// TIA Portal V17 export
// export: Created 2024-06-16T17:47:20.4638642Z, ExportSetting WithDefaults, DisplayName Totally Integrated Automation Portal, DisplayVersion V17, DisplayName TIA Portal Openness, DisplayVersion V17, DisplayName TIA Portal Version Control Interface, DisplayVersion V17, DisplayName STEP 7 Professional, DisplayVersion V17, DisplayName STEP 7 Safety, DisplayVersion V17, DisplayName WinCC Professional, DisplayVersion V17
FUNCTION "Manager" : Void   // FC1, LAD
{ S7_Optimized_Access := 'TRUE' }
VERSION : 0.1
// stored: AutoNumber false, IsIECCheckEnabled false, SetENOAutomatically false, UDAEnableTagReadback false
BEGIN

REGION Network 1
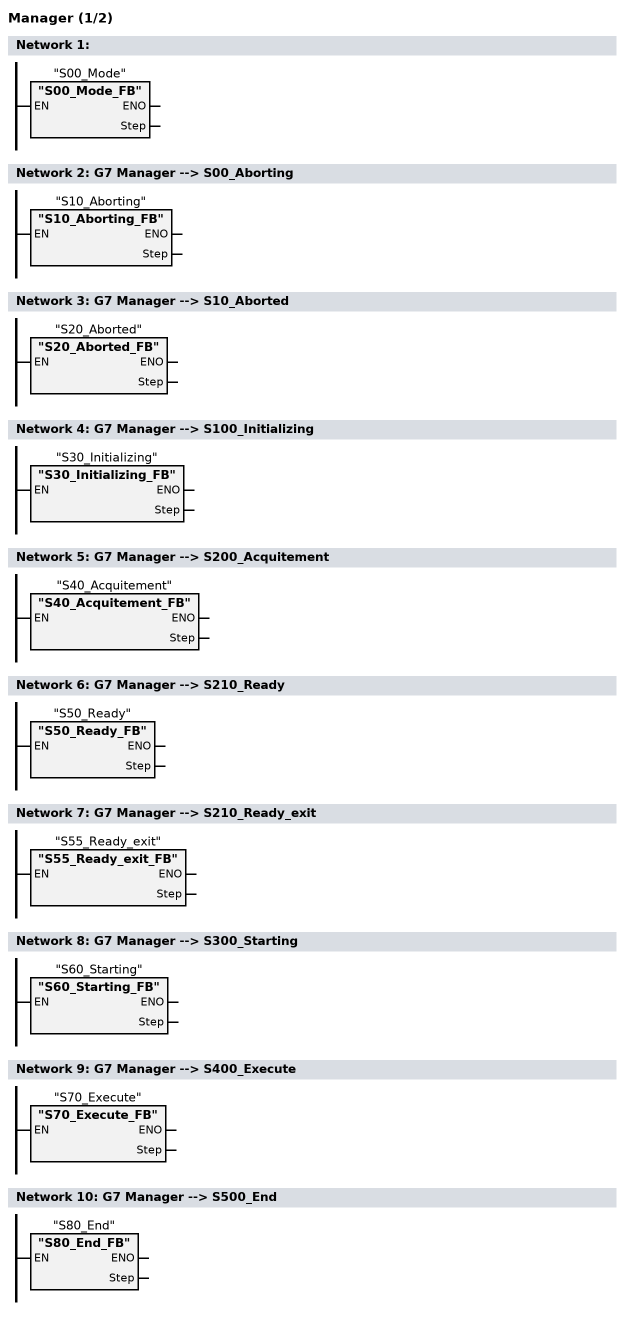
   RUNG wire#powerrail
      "S00_Mode"("Step" =>)
   END_RUNG
   // the same network as SCL:
   "S00_Mode"();   // "S00_Mode_FB"
END_REGION

REGION Network 2: G7 Manager --> S00_Aborting
   RUNG wire#powerrail
      "S10_Aborting"("Step" =>)
   END_RUNG
   // the same network as SCL:
   "S10_Aborting"();   // "S10_Aborting_FB"
END_REGION

REGION Network 3: G7 Manager --> S10_Aborted
   RUNG wire#powerrail
      "S20_Aborted"("Step" =>)
   END_RUNG
   // the same network as SCL:
   "S20_Aborted"();   // "S20_Aborted_FB"
END_REGION

REGION Network 4: G7 Manager --> S100_Initializing
   RUNG wire#powerrail
      "S30_Initializing"("Step" =>)
   END_RUNG
   // the same network as SCL:
   "S30_Initializing"();   // "S30_Initializing_FB"
END_REGION

REGION Network 5: G7 Manager --> S200_Acquitement
   RUNG wire#powerrail
      "S40_Acquitement"("Step" =>)
   END_RUNG
   // the same network as SCL:
   "S40_Acquitement"();   // "S40_Acquitement_FB"
END_REGION

REGION Network 6: G7 Manager --> S210_Ready
   RUNG wire#powerrail
      "S50_Ready"("Step" =>)
   END_RUNG
   // the same network as SCL:
   "S50_Ready"();   // "S50_Ready_FB"
END_REGION

REGION Network 7: G7 Manager --> S210_Ready_exit
   RUNG wire#powerrail
      "S55_Ready_exit"("Step" =>)
   END_RUNG
   // the same network as SCL:
   "S55_Ready_exit"();   // "S55_Ready_exit_FB"
END_REGION

REGION Network 8: G7 Manager --> S300_Starting
   RUNG wire#powerrail
      "S60_Starting"("Step" =>)
   END_RUNG
   // the same network as SCL:
   "S60_Starting"();   // "S60_Starting_FB"
END_REGION

REGION Network 9: G7 Manager --> S400_Execute
   RUNG wire#powerrail
      "S70_Execute"("Step" =>)
   END_RUNG
   // the same network as SCL:
   "S70_Execute"();   // "S70_Execute_FB"
END_REGION

REGION Network 10: G7 Manager --> S500_End
   RUNG wire#powerrail
      "S80_End"("Step" =>)
   END_RUNG
   // the same network as SCL:
   "S80_End"();   // "S80_End_FB"
END_REGION

REGION Network 11: G7 Manager --> S600_Stopping
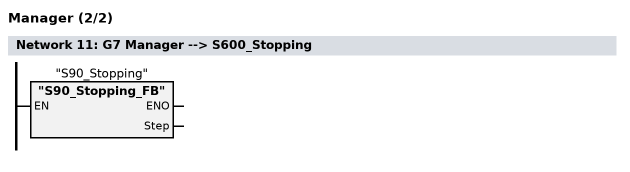
   RUNG wire#powerrail
      "S90_Stopping"("Step" =>)
   END_RUNG
   // the same network as SCL:
   "S90_Stopping"();   // "S90_Stopping_FB"
END_REGION
END_FUNCTION
